FUNCTION_BLOCK AutoMove2
VAR_INPUT
END_VAR
VAR_OUTPUT
END_VAR
VAR
	Target : POZAYZ;
END_VAR

IF AUTO.StageSelect > 0 AND AUTO.StageSelect < AUTO.StageMax THEN
	IF AUTO.Stages[AUTO.Recept][Auto.StageSelect].I = 0 THEN
		Target := AUTO.Positions[AUTO.Stages[AUTO.Recept][Auto.StageSelect].T];
		IF AUTO.Current.Z <> Target.Z  THEN
		AUTO.MotorIzbira := 1;
		IF AUTO.Current.Z > Target.Z THEN
			AUTO.VrtenjeSmer := TRUE;
		ELSE
			AUTO.VrtenjeSmer := FALSE;
		END_IF
		AUTO.VrtenjePremik := TRUE;
	ELSIF AUTO.Current.Y <> Target.Y  THEN
		AUTO.MotorIzbira := 3;
		IF AUTO.Current.Y > Target.Y THEN
			AUTO.IztegSmer := TRUE;
		ELSE
			AUTO.IztegSmer := FALSE;
		END_IF
		AUTO.IztegPremik := TRUE;
	ELSIF AUTO.Current.A <> Target.A  THEN
		AUTO.MotorIzbira := 2;
		IF AUTO.Current.A > Target.A THEN
			AUTO.DvigSmer := TRUE;
		ELSE
			AUTO.DvigSmer := FALSE;
		END_IF
		AUTO.DvigPremik := TRUE;
	ELSIF AUTO.Current.P <> AUTO.Stages[AUTO.Recept][Auto.StageSelect].P  THEN
		AUTO.MotorIzbira := 4;
		IF AUTO.Current.P > AUTO.Stages[AUTO.Recept][Auto.StageSelect].P THEN
			AUTO.PrijemSmer := TRUE;
		ELSE
			AUTO.PrijemSmer := FALSE;
		END_IF
		AUTO.PrijemPremik := TRUE;
	ELSE
		AUTO.VrtenjePremik := FALSE;
		AUTO.DvigPremik := FALSE;
		AUTO.IztegPremik := FALSE;
		AUTO.PrijemPremik := FALSE;
		AUTO.StageSelect := AUTO.StageSelect + 1;
	END_IF
	ELSE
		Target := AUTO.Items[AUTO.Stages[AUTO.Recept][Auto.StageSelect].I];
		IF AUTO.Current.A <> Target.A  THEN
		AUTO.MotorIzbira := 1;
		IF AUTO.Current.A > Target.A THEN
			AUTO.VrtenjeSmer := TRUE;
		ELSE
			AUTO.VrtenjeSmer := FALSE;
		END_IF
		AUTO.VrtenjePremik := TRUE;
	ELSIF AUTO.Current.Y <> Target.Y  THEN
		AUTO.MotorIzbira := 3;
		IF AUTO.Current.Y > Target.Y THEN
			AUTO.IztegSmer := TRUE;
		ELSE
			AUTO.IztegSmer := FALSE;
		END_IF
		AUTO.IztegPremik := TRUE;
	ELSIF AUTO.Current.Z <> Target.Z  THEN
		AUTO.MotorIzbira := 2;
		IF AUTO.Current.Z > Target.Z THEN
			AUTO.DvigSmer := TRUE;
		ELSE
			AUTO.DvigSmer := FALSE;
		END_IF
		AUTO.DvigPremik := TRUE;
	ELSIF AUTO.Current.P <> AUTO.Stages[AUTO.Recept][Auto.StageSelect].P  THEN
		AUTO.MotorIzbira := 4;
		IF AUTO.Current.P > AUTO.Stages[AUTO.Recept][Auto.StageSelect].P THEN
			AUTO.PrijemSmer := TRUE;
		ELSE
			AUTO.PrijemSmer := FALSE;
		END_IF
		AUTO.PrijemPremik := TRUE;
	ELSE
		AUTO.VrtenjePremik := FALSE;
		AUTO.DvigPremik := FALSE;
		AUTO.IztegPremik := FALSE;
		AUTO.PrijemPremik := FALSE;
		AUTO.StageSelect := AUTO.StageSelect + 1;
	END_IF
	END_IF
	
END_IF

END_FUNCTION_BLOCK

(* stored: Version 1.1.0.1, ProductVersion 3.1.4024.12
   POU AutoMove2: Id {aacb6a7f-e5c4-4e38-9ad4-dc662886ab74}, SpecialFunc None *)
